// TIA Portal V17 export
FUNCTION "烧嘴报警" : Void   // FC, LAD
{ S7_Optimized_Access := 'TRUE' }
VERSION : 0.1
// stored: AutoNumber true, IsIECCheckEnabled false, SetENOAutomatically false
BEGIN

REGION Network 1
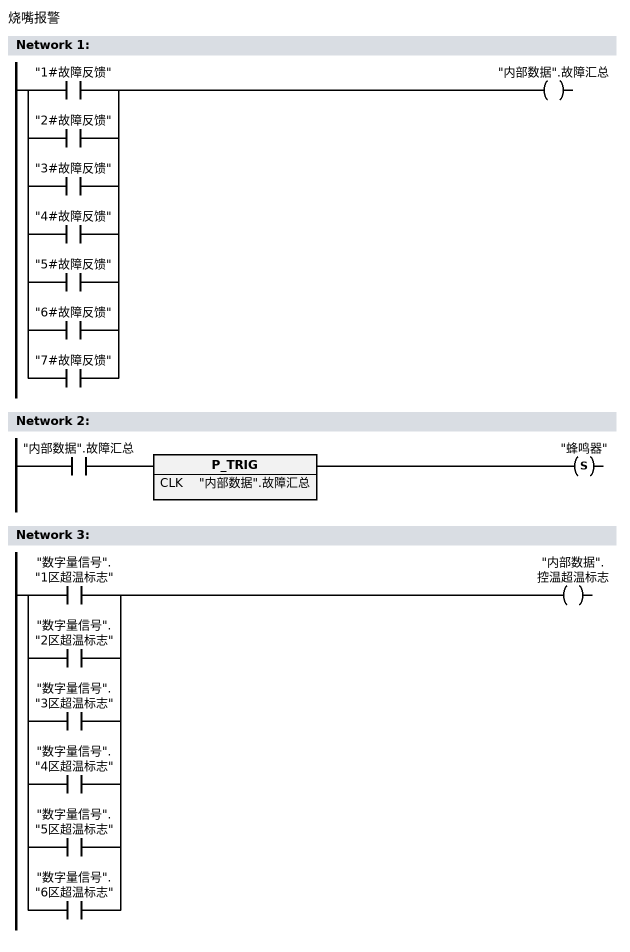
   RUNG wire#powerrail
      Contact( "1#故障反馈" )
      wire#w1
      wire#w2
      Coil( "内部数据".故障汇总 )
   END_RUNG
   RUNG wire#powerrail
      Contact( "2#故障反馈" )
   END_RUNG wire#w1
   RUNG wire#powerrail
      Contact( "3#故障反馈" )
   END_RUNG wire#w1
   RUNG wire#powerrail
      Contact( "4#故障反馈" )
   END_RUNG wire#w1
   RUNG wire#powerrail
      Contact( "5#故障反馈" )
      wire#w3
   END_RUNG wire#w2
   RUNG wire#powerrail
      Contact( "6#故障反馈" )
   END_RUNG wire#w3
   RUNG wire#powerrail
      Contact( "7#故障反馈" )
   END_RUNG wire#w3
   // the same network as SCL:
   "内部数据".故障汇总 := "1#故障反馈" OR "2#故障反馈" OR "3#故障反馈" OR "4#故障反馈" OR "5#故障反馈" OR "6#故障反馈" OR "7#故障反馈";
END_REGION

REGION Network 2
   // no checked SCL form for this network; see the picture
END_REGION

REGION Network 3
   RUNG wire#powerrail
      Contact( "数字量信号"."1区超温标志" )
      wire#w1
      wire#w2
      Coil( "内部数据".控温超温标志 )
   END_RUNG
   RUNG wire#powerrail
      Contact( "数字量信号"."2区超温标志" )
   END_RUNG wire#w1
   RUNG wire#powerrail
      Contact( "数字量信号"."3区超温标志" )
   END_RUNG wire#w1
   RUNG wire#powerrail
      Contact( "数字量信号"."4区超温标志" )
      wire#w3
   END_RUNG wire#w2
   RUNG wire#powerrail
      Contact( "数字量信号"."5区超温标志" )
   END_RUNG wire#w3
   RUNG wire#powerrail
      Contact( "数字量信号"."6区超温标志" )
   END_RUNG wire#w3
   // the same network as SCL:
   "内部数据".控温超温标志 := "数字量信号"."1区超温标志" OR "数字量信号"."2区超温标志" OR "数字量信号"."3区超温标志" OR "数字量信号"."4区超温标志" OR "数字量信号"."5区超温标志" OR "数字量信号"."6区超温标志";
END_REGION
END_FUNCTION
